Staubli VAL3: teachPoint.pgx

public program teachPoint(string x_sPointName, tool x_tTool, frame x_fFrame, point& x_pPoint)
  local string l_sTemp
  local num l_nNum
  local point l_pPoint
begin

  wait(getKey()==-1)

  userPage()
  call clrscr()

  l_sTemp = "teaching "+x_sPointName
  call sCenterTitle(l_sTemp)

  title(l_sTemp)

  gotoxy(0,4)
  l_sTemp = "premi F8 per acquisire "+x_sPointName
  call sCenterRow(l_sTemp)
  putln(l_sTemp)

  gotoxy(0,5)
  l_sTemp = "premi F1 per uscire"
  call sCenterRow(l_sTemp)
  putln(l_sTemp)

  gotoxy(0,13)
  put("F1=Esc")
  gotoxy(34,13)
  put("F8=Qui")

  do
    l_nNum=get()
    if l_nNum==271
      call dialogOnlyOK("teaching "+x_sPointName,"acquisizione punto annullata",x_sPointName+" non è stato modificato","premi F1 per continuare","")
    elseIf l_nNum==278
      l_pPoint = here(x_tTool, x_fFrame)
      x_pPoint.trsf = position(l_pPoint, x_fFrame)
      call trsfDialogIns("teaching "+x_sPointName, "", x_pPoint.trsf)
    endIf
  until l_nNum==271 or l_nNum==278

  call clrscr()

  wait(getKey()==-1)

end
